FUNCTION_BLOCK EL3312
VAR
	_io : EL3xx2_Data;
	{attribute addProperty Name "WcState"}
	_wcState : WcStateInputToggle;
	{attribute addProperty Name "Info data"}
	_infoData : InfoDataAds;
END_VAR

PROPERTY IO : REFERENCE TO EL3xx2_Data
GET
IO REF= _io;
END_GET
END_PROPERTY

PROPERTY WcState : REFERENCE TO WcStateInputToggle
GET
WcState REF= _wcState;
END_GET
END_PROPERTY

END_FUNCTION_BLOCK

(* stored: Version 1.1.0.1, ProductVersion 3.1.4024.9
   POU EL3312: Id {d1caf4c3-db1d-060e-2b3c-a8ee3432d409}, SpecialFunc None
   Property IO: Id {1dc4ff80-9333-0a6f-3264-2ed14e60850b}
   Get Get: Id {de0809b0-ac6d-0301-303a-ada3a13383f8}
   Property WcState: Id {aed048de-9ade-0dbd-06f6-1521cc9cd674}
   Get Get: Id {2493494e-f353-0f07-10a6-d66f76f823ac} *)
